# EPICS IOC start-up script: ioc_startup_example.iocsh
#- require the ECMC_AGIR module
#- this calls ${ECMC_AGIR_DIR}startup.cmd, which in turn pulls together all dependencies
require ECMC_AGIR, IBS

#- instantiate girder
#- DEV = AGIR-TEST
#- Synchronization ON
#- HomeOffsets for prototype-rig in OTLA
runScript $(ECMC_AGIR_DIR)/addGirder.iocsh, "DEV='AGIR-TEST',Synchronization=True,HO_TY1=-19.71609,HO_TY2=-29.68623,HO_TX1=2.42422,HO_TX2=0.70461"
